PROGRAM OP130_AutoSequence
VAR
	State: INT;
	OP130_Stepper_Pos : REAL:=24;
	temp5: BOOL;
	OP130_StnEnableTRIG: R_TRIG;
	dry_run:BOOL;
	fix_lh:INT;
	fix_rh:INT;
	op130_clamp_stepper_work: BOOL;
	op130_cycle_time_fb :FB_cycleTime;
	OP130_Cycle_time : UDINT;
	parts_ok: INT;
	parts_nok: INT;
END_VAR

IF (NOT OP130_Auto OR  OP130_ErrorActive OR OP130_HomeRunning OR OP130_Machine_Stop ) THEN
	OP130_GVL.OP130_AutoRunning:= FALSE;
	OP130_GVL.OP130_Home_ConditionOK:=FALSE;
	OP130_Dry_Run:=FALSE;
	OP130_ComponentOk:=FALSE;
	OP130_ComponentNok:=FALSE;
	OP130_RH_Comp_OK:=FALSE;
	OP130_RH_Comp_NOK:= FALSE;
	OP130_LH_Comp_OK:=FALSE;
	OP130_LH_Comp_NOK:= FALSE;
	OP130_AutoSeq:= 10;
	OP130_LH_AutoSeq:=0;
	OP130_RH_AutoSeq:=0;
END_IF

(*IF OP130_Auto AND NOT OP130_HomeRunning THEN
	SR130_Stepper_Control.Position:=OP130_Stepper_Pos;
	SR130_Stepper_Control.Velocity:=50;
ELSE
	SR130_Stepper_Control.Position:=0;
	SR130_Stepper_Control.Velocity:=50;
	SR130_Stepper_Control.ABSmove_Start:=1;
END_IF
*)

CASE OP130_AutoSeq OF 
	10:IF (OP130_Auto) THEN		// Check Automode Selected
		  OP130_AutoSeq :=20;
	    END_IF
		
	20:IF ( NOT OP130_ErrorActive) THEN		//Check No error
		  OP130_AutoSeq:=30;
	   END_IF
	   
	30:IF (NOT OP130_HomeRunning) THEN		//Check No Homerunning
		  OP130_AutoSeq :=40;
		END_IF
		
    40:IF ( OP130_GVL.OP130_Temp_Home_OK)THEN	//Check Machine in Home
		  OP130_AutoSeq:= 50;
		END_IF
		
	50:IF ( NOT OP130_OperationCompleted) THEN		// Check Operation Completed Reset
		OP130_AutoSeq:=60;
		END_IF
		
	60:IF (NOT OP130_ComponentOk) THEN		// Check Component Ok Reset
		OP130_AutoSeq:=70;
		END_IF
		
	70:IF (NOT OP130_ComponentNok) THEN 	// Check Component NOk Reset
		OP130_AutoSeq:= 120;
		END_IF
		
    120:IF  (OP130_HMI_Cycle_Start OR OP130_Dry_Run) THEN		//Machine Start in Fully Automatic or Press Cycle Start For Semi Automatic
		    OP130_GVL.OP130_Home_ConditionOK:=TRUE;
	 			IF( OP130_GVL.OP130_Home_ConditionOK AND OP130_AutoSelected) THEN
					OP130_AutoRunning:=TRUE;
					OP130_StepRunning:= FALSE;
				
				ELSIF (OP130_Home_ConditionOK AND OP130_StepSelected) THEN
					OP130_AutoRunning:=FALSE;
					OP130_StepRunning:= TRUE;
				END_IF;
		 END_IF
		 IF ((OP130_AutoRunning OR OP130_StepRunning) AND OP130_StartEnable) THEN
			     SR130_Stepper_Control.ABSmove_Start:=1;
				 OP130_AutoSeq:= 130;
		END_IF
	130:IF (OP130_StartEnable) THEN // Check Previous Station Completed
				OP130_AutoSeq:= 131;       
     	END_IF
	
     131:   SR130_Stepper_Control.Position:=88;
            SR130_Stepper_Control.Velocity:=50;
		    SR130_Stepper_Control.ABSmove_Start:=TRUE;
             IF SR130_Clm_Stepper.bAxisInPosition AND op130_clamp_stepper_work THEN
				SR130_Stepper_Control.ABSmove_Start:=FALSE; 
		        OP130_AutoSeq:= 140;
		     END_IF
	 	
	140: IF NOT OP130_STN_ENABLE AND MOVER_POS_RECHED[OP130_STN_MOVER] AND fix_lh <> 120 AND fix_rh <> 120 THEN
         	OP130_AutoSeq:= 200;
         ELSIF OP130_STN_ENABLE AND fix_lh =120 AND fix_rh =120 THEN
           OP130_Prev_LH_COMP_OK:=TRUE;
	       OP130_Prev_RH_COMP_OK:=TRUE;
           OP130_Prev_LH_COMP_NOK:=FALSE;
           OP130_Prev_RH_COMP_NOK:=FALSE;
		   OP130_AutoSeq:= 141;
         ELSIF OP130_STN_ENABLE AND fix_lh = 120 AND fix_rh =121 THEN
           OP130_Prev_LH_COMP_OK:=TRUE;
	       OP130_Prev_RH_COMP_OK:=FALSE;
           OP130_Prev_LH_COMP_NOK:=FALSE;
           OP130_Prev_RH_COMP_NOK:=TRUE;
		   OP130_AutoSeq:= 141;
         ELSIF OP130_STN_ENABLE AND fix_lh = 121 AND fix_rh =120 THEN
           OP130_Prev_LH_COMP_OK:=false;
	       OP130_Prev_RH_COMP_OK:=TRUE;
		   OP130_Prev_LH_COMP_NOK:=TRUE;
           OP130_Prev_RH_COMP_NOK:=FALSE;
           OP130_AutoSeq:= 141;
          END_IF 
		  
    141:	OP130_LH_AutoSeq:=10;
            OP130_RH_AutoSeq:=10;
		    OP130_AutoSeq:= 150;  
		  
   
	150:IF (OP130_LH_Operation_Completed AND OP130_RH_Operation_Completed ) THEN	//Waiting For Both RH & LH Seq Completion
			OP130_MVR_DN_PERMISSION			:= TRUE;
			OP130_AutoSeq					:= 151;			
		 END_IF
		 OP130_CURR_MOVER		:=OP130_STN_MOVER;
	
	151: IF NOT OP130_MVR_DN_PERMISSION THEN
			OP130_AutoSeq					:= 155;		
		END_IF	 
	
	155:IF OP130_LH_Comp_OK AND OP130_rH_Comp_OK THEN
				MOVER_CMP_STATUS[OP130_CURR_MOVER][1]:=130;	
                MOVER_CMP_STATUS[OP130_CURR_MOVER][2]:=130;
		            IF MOVER_CMP_STATUS[OP130_CURR_MOVER][1]=130 AND MOVER_CMP_STATUS[OP130_CURR_MOVER][2]=130 THEN
			     	STATION_DONE[OP130_CURR_MOVER][OP130_XTS_POS_NO]			:= TRUE;
			            OP130_AutoSeq:= 160;
						parts_ok :=parts_ok+1;
				     END_IF
				ELSIF OP130_LH_Comp_NOK AND OP130_rH_Comp_OK THEN	
					  MOVER_CMP_STATUS[OP130_CURR_MOVER][1]:=130;	
                      MOVER_CMP_STATUS[OP130_CURR_MOVER][2]:=130;
		               IF MOVER_CMP_STATUS[OP130_CURR_MOVER][1]=130 AND MOVER_CMP_STATUS[OP130_CURR_MOVER][2]=130 THEN
			         	STATION_DONE[OP130_CURR_MOVER][OP130_XTS_POS_NO]			:= TRUE;
			              OP130_AutoSeq:= 160;
						  parts_nok :=parts_nok+1;
			    	   END_IF
                 ELSIF OP130_LH_Comp_OK AND OP130_rH_Comp_NOK THEN	
					  MOVER_CMP_STATUS[OP130_CURR_MOVER][1]:=130;	
                      MOVER_CMP_STATUS[OP130_CURR_MOVER][2]:=130;
		               IF MOVER_CMP_STATUS[OP130_CURR_MOVER][1]=130 AND MOVER_CMP_STATUS[OP130_CURR_MOVER][2]=130 THEN
			       	STATION_DONE[OP130_CURR_MOVER][OP130_XTS_POS_NO]			:= TRUE;
			              OP130_AutoSeq:= 160;
						  parts_nok :=parts_nok+1;
			    	   END_IF	
					   ELSIF OP130_LH_Comp_NOK AND OP130_rH_Comp_NOK THEN	
					  MOVER_CMP_STATUS[OP130_CURR_MOVER][1]         :=130;	
                      MOVER_CMP_STATUS[OP130_CURR_MOVER][2]         :=130;
		               IF MOVER_CMP_STATUS[OP130_CURR_MOVER][1]=130 AND MOVER_CMP_STATUS[OP130_CURR_MOVER][2]=130 THEN
			          	STATION_DONE[OP130_CURR_MOVER][OP130_XTS_POS_NO]			:= TRUE;
			              OP130_AutoSeq:= 160;
						  parts_nok :=parts_nok+1;
					   END_IF
			  END_IF	
		
	160:IF ( OP130_StartEnable) THEN  // Operation Completed
	        OP130_Cycle_Time_Stop                                   :=TRUE;
			OP130_OperationCompleted                                :=TRUE;
			OP130_AutoSeq                                           := 170;
			STATION_DONE[OP130_CURR_MOVER][OP130_XTS_POS_NO]			:= TRUE;
		END_IF
		
	170:OP130_LH_Operation_Completed             :=FALSE;
	    OP130_RH_Operation_Completed             :=FALSE;
	    OP130_OperationCompleted                 :=FALSE;
	    OP130_ComponentOk                        :=FALSE;
	    OP130_ComponentNOk                       :=FALSE;
	    OP130_AutoSeq                            :=180;
	
	(*171 : SR130_Stepper_Control.Position:=0;
          SR130_Stepper_Control.Velocity:=50;
		  SR130_Stepper_Control.ABSmove_Start:=TRUE;
		  
             IF SR130_Clm_Stepper.bAxisInPosition THEN
				SR130_Stepper_Control.ABSmove_Start:=FALSE; 
		        OP130_AutoSeq:= 180;
		     END_IF*)
	
	180:		// Reset All Bits	
	
        OP130_Prev_LH_COMP_OK:=FALSE;
		OP130_Prev_RH_COMP_OK:=FALSE;						
        OP130_LH_Comp_OK:=FALSE;
        OP130_LH_Comp_NOK:=FALSE;
        OP130_RH_Comp_OK:=FALSE;
        OP130_RH_Comp_NOK:=FALSE;
        OP130_LH_AutoSeq:=0;
		OP130_RH_AutoSeq:=0;
		OP130_AutoSeq:= 130;
		
		
   200:	MOVER_CMP_STATUS[OP130_CURR_MOVER][1]:=130;	 ///// NEED TO BE UPDATED AS 131
        MOVER_CMP_STATUS[OP130_CURR_MOVER][2]:=130;
		IF MOVER_CMP_STATUS[OP130_CURR_MOVER][1]=130 AND MOVER_CMP_STATUS[OP130_CURR_MOVER][2]=130 THEN
				STATION_DONE[OP130_CURR_MOVER][OP130_XTS_POS_NO]			:= TRUE;
			OP130_AutoSeq:= 180;
		END_IF


END_CASE

op130_cycle_time_fb(i_b_startTime:=OP130_STN_ENABLE , i_b_stopTime:= NOT OP130_STN_ENABLE , o_t_StationTime=>OP130_Cycle_time );
dry_run:=All_Station_Dry_Run;
//staus FOR movers 
IF  dry_run THEN
	fix_lh :=120;
	fix_rh :=120;
ELSE 
	fix_lh := MOVER_CMP_STATUS[OP130_STN_MOVER][1];
	fix_rh := MOVER_CMP_STATUS[OP130_STN_MOVER][2];
END_IF

op130_clamp_stepper_work:=In_Range(value:=SR130_Clm_Stepper.Actual_position, setvalue:= 88, tolerance:= 0.2);



//############################		OP130 STATION ENABLE CONDITION		##########################

	OP130_STN_MOVER					:= MOVER_POSITION[OP130_XTS_POS_NO];
	IF AUTO_WITH_XTS THEN
	IF OP130_STN_MOVER>0 THEN
	IF NOT(END_OF_CYCLE AND MOVER_CMP_STATUS[OP130_STN_MOVER][1]=5 AND MOVER_CMP_STATUS[OP130_STN_MOVER][2]=5)THEN		
	OP130_STN_ENABLE				:= MOVER_POS_RECHED[OP130_STN_MOVER] AND ((MOVER_CMP_STATUS[OP130_STN_MOVER][1]=120)OR 
										(MOVER_CMP_STATUS[OP130_STN_MOVER][2]=120))AND STATION_ENABLE_CONTROL;		
	ELSE
	STATION_DONE[OP130_STN_MOVER][OP130_XTS_POS_NO]			:= TRUE;		
	END_IF
	ELSE
	OP130_STN_ENABLE				:= FALSE;	
	END_IF
	END_IF

END_PROGRAM

(* stored: Version 1.1.0.1, ProductVersion 3.1.4024.11
   POU OP130_AutoSequence: Id {e3c04423-5f32-4fad-aa6c-d4f0af15e254}, SpecialFunc None *)
